(* Logix 5000 project; controller Add_On_MIG Emulate 5570 rev 36.11; software revision 36.00 *)

TASK MainTask (continuous, watchdog 500 ms) : MainProgram, Model

MODULES
   Local : Emulate 5570 (ICP 2, rev 36.11)
       : 1756-IB16 (ICP 3, rev 3.1, Input RPI 20 ms)
       : vendor 1 type 7 code 16 (ICP 4, rev 3.1, Output RPI 20 ms)
END_MODULES

ADD_ON_INSTRUCTION MIG_Interface   (* revision 1.0 *)
VAR_INPUT
   Arc_Start : BOOL; {required}   // Begin MIG Welding
   Arc_End : BOOL; {required}   // MIG Welding Finished
END_VAR
VAR_OUTPUT
   Wire_Feed : BOOL; {access None, required}   // Energize Filler Wire Feeder
   Gas_Flow : BOOL; {access Read Only, required}   // Open Shielding Gas Valve
   Arc_On : BOOL; {access Read Only, required}   // MIG Arc Established
END_VAR
VAR_INPUT
   Pre_Weld_Delay : DINT; {required}   // Gas and Wire Preflow
   Fault_Arc : BOOL; {required}   // Loss of MIG Welding Arc
   Fault_Wire : BOOL; {required}   // Wire feed not detected
END_VAR
VAR
   BOR_01 : FBD_BOOLEAN_OR; {access None}
   BAND_01 : FBD_BOOLEAN_AND := (In1 := 1, In2 := 1, In3 := 1, In4 := 1, In5 := 1, In6 := 1, In7 := 1, In8 := 1); {access None}
   TONR_01 : FBD_TIMER; {access None}
   BNOT_01 : FBD_BOOLEAN_NOT := (In := 1); {access None}
   __lF7E3A54EB71210EA : BOOL; {access None}
   __lF6B7A888152192F8 : BOOL; {access None}
   __l7528BC9BE018A205 : BOOL; {access None}
   __l896FE0D45DD24A0F : BOOL; {access None}
   __l6A81249255479518 : DINT; {access None}
END_VAR

ROUTINE Logic   (* function block diagram *)
   SHEET 1
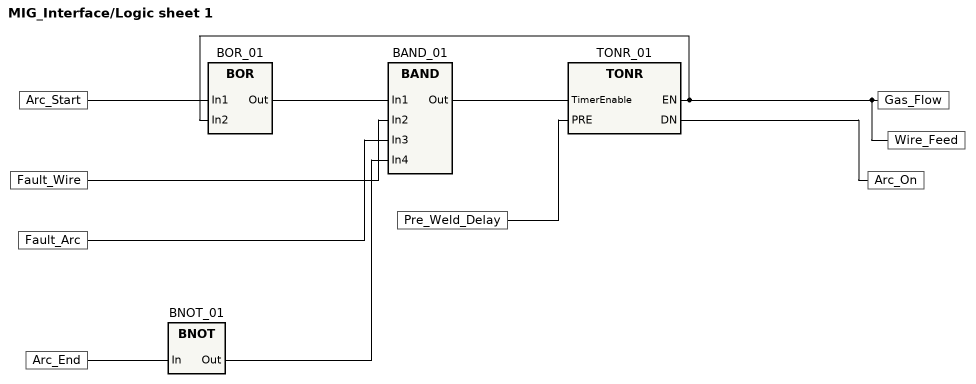
   BNOT_01 : BNOT(In := Arc_End);
   BOR_01 : BOR(In1 := Arc_Start, In2 := TONR_01.EN {feedback});
   BAND_01 : BAND(In1 := BOR_01.Out, In2 := Fault_Wire, In3 := Fault_Arc, In4 := BNOT_01.Out);
   TONR_01 : TONR(TimerEnable := BAND_01.Out, PRE := Pre_Weld_Delay);
   Arc_On := TONR_01.DN;
   Gas_Flow := TONR_01.EN;
   Wire_Feed := TONR_01.EN;
END_ROUTINE
END_ADD_ON_INSTRUCTION

PROGRAM MainProgram   (* main routine MainRoutine *)
VAR
   Welder1 : MIG_Interface := (Pre_Weld_Delay := 10000);   // MIG Welding Station No. 1
   Welder2 : MIG_Interface;   // MIG Welding Station Nno. 2
END_VAR

ROUTINE MainRoutine   (* ladder *)
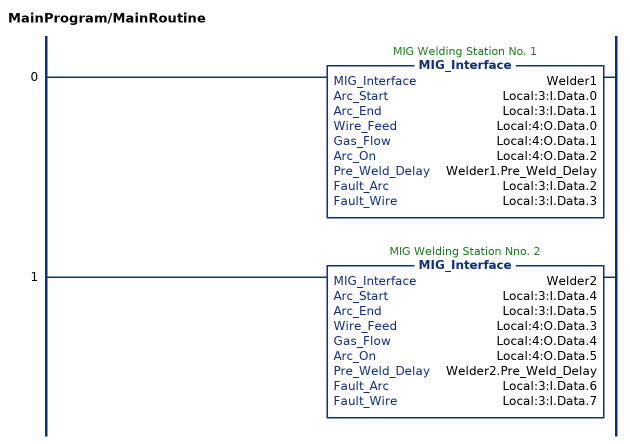
   0: MIG_Interface(Welder1,Local:3:I.Data.0,Local:3:I.Data.1,Local:4:O.Data.0,Local:4:O.Data.1,Local:4:O.Data.2,Welder1.Pre_Weld_Delay,Local:3:I.Data.2,Local:3:I.Data.3);
   1: MIG_Interface(Welder2,Local:3:I.Data.4,Local:3:I.Data.5,Local:4:O.Data.3,Local:4:O.Data.4,Local:4:O.Data.5,Welder2.Pre_Weld_Delay,Local:3:I.Data.6,Local:3:I.Data.7);
END_ROUTINE
END_PROGRAM

PROGRAM Model   (* main routine Emulation *)
VAR
   Welder1_End : BOOL;
   Welder1_Fault_Arc : BOOL;
   Welder1_Fault_Wire : BOOL;
   Welder1_Start : BOOL;
   Welder2_End : BOOL;
   Welder2_Fault_Arc : BOOL;
   Welder2_Fault_Wire : BOOL;
   Welder2_Start : BOOL;
END_VAR

ROUTINE Emulation   (* ladder *)
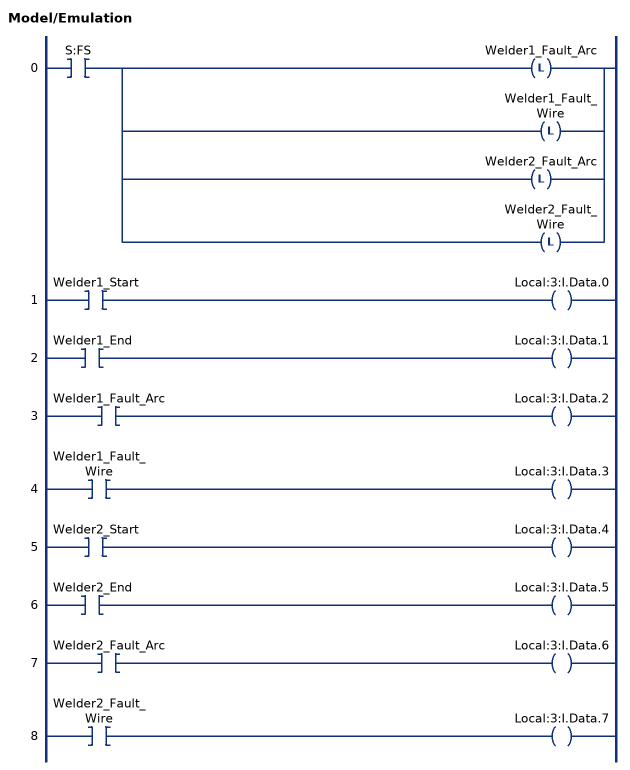
   0: XIC(S:FS)[OTL(Welder1_Fault_Arc) ,OTL(Welder1_Fault_Wire) ,OTL(Welder2_Fault_Arc) ,OTL(Welder2_Fault_Wire) ];
   1: XIC(Welder1_Start)OTE(Local:3:I.Data.0);
   2: XIC(Welder1_End)OTE(Local:3:I.Data.1);
   3: XIC(Welder1_Fault_Arc)OTE(Local:3:I.Data.2);
   4: XIC(Welder1_Fault_Wire)OTE(Local:3:I.Data.3);
   5: XIC(Welder2_Start)OTE(Local:3:I.Data.4);
   6: XIC(Welder2_End)OTE(Local:3:I.Data.5);
   7: XIC(Welder2_Fault_Arc)OTE(Local:3:I.Data.6);
   8: XIC(Welder2_Fault_Wire)OTE(Local:3:I.Data.7);
END_ROUTINE
END_PROGRAM
